Universal Robots PolyScope program: rtde_control_loop_new.urp

Program rtde_control_loop_new (installation=default directory=/programs createdIn=3.2.19275.0 lastSavedIn=5.4.0.76181 robotSerialNumber=20195500451)
Calibrated DH parameters: a=[0.00002, -0.231658, -0.317125, 0.000011, 0.000055, 0]; d=[0.162082, 123.190176, -180.284242, 57.22734, 0.099524, 0.09934]; alpha=[1.569304, 0.00289, 0.004025, 1.569925, -1.569026, 0]; deltaTheta=[0, 0.993923, 4.662183, 0.627072, 0.000001, 0]
BeforeStart
  setp := [0,0,0,0,0,0]
  setj := [0,0,0,0,0,0]
  moving := 0
  blocking := 0.008
  lookahead := 0.03
  gain := 500
  maxPosError := 0.01
  maxOrientError := 0.01
  Set NoAction (payload=0.2 tcpAsCog=false)
  SuppressedNode
    Script: position_deviation_warning(True)
Robot Program (runOnlyOnce=false)
  Script: write_output_integer_register(0, 0)
  If moving == 1
    Script: servoj(setj,0,0,blocking,lookahead,gain)
  ElseIf moving == 2
    Script: speedj(setp,gain,blocking)
  ElseIf moving == 3
    Script: movej(setp,gain,maxPosError,blocking,maxOrientError)
  ElseIf moving == 4
    Script: movel(setp,gain,maxPosError,blocking,maxOrientError)
  ElseIf moving == 5
    Script: force_mode(Base,[1,1,0,0,0,0],[10*sin(time_start),0,0,0,0,0],2,[2,2,2,0.1,0.1,0.1])
  Script: sync()
Thread Thread_1 (runOnlyOnce=false trackProgramExecution=false)
  setj := [0,0,0,0,0,0]
  setp := [0,0,0,0,0,0]
  moving := 0
  blocking := 0.008
  lookahead := 0.03
  gain := 500
  maxPosError := 0.01
  maxOrientError := 0.01
  Loop Forever
    tmp := [0,0,0,0,0,0,0,0,0,0,0,0]
    Script: tmp[0] = read_input_float_register(0)
    Script: tmp[1] = read_input_float_register(1)
    Script: tmp[2] = read_input_float_register(2)
    Script: tmp[3] = read_input_float_register(3)
    Script: tmp[4] = read_input_float_register(4)
    Script: tmp[5] = read_input_float_register(5)
    Script: tmp[6] = read_input_float_register(6)
    Script: tmp[7] = read_input_float_register(7)
    Script: tmp[8] = read_input_float_register(8)
    Script: tmp[9] = read_input_float_register(9)
    Script: tmp[10] = read_input_float_register(10)
    Script: tmp[11] = read_input_float_register(11)
    If tmp != [0,0,0,0,0,0,0,0,0,0,0,0]
      moving := tmp[6]
      blocking := tmp[7]
      lookahead := tmp[8]
      gain := tmp[9]
      maxPosError := tmp[10]
      maxOrientError := tmp[11]
      If moving == 1
        setj := [tmp[0],tmp[1],tmp[2],tmp[3],tmp[4],tmp[5]]
      ElseIf moving == 2
        setp := [tmp[0],tmp[1],tmp[2],tmp[3],tmp[4],tmp[5]]
    Script: sync()
